FUNCTION_BLOCK TaskGUIFB (* JADE WORKER *)
  (* Standard: 61499-1 *)
  (* Version 1.0, 2014-04-22, Ahmed, Fraunhofer IGD *)
  (* Compiler header: package fb.gui; *)
  (* Compiler Java Sun JDK 1.5.0 *)
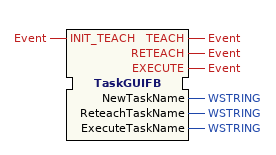
  EVENT_INPUT
    INIT_TEACH;
  END_EVENT
  EVENT_OUTPUT
    TEACH;
    RETEACH;
    EXECUTE;
  END_EVENT
  VAR_OUTPUT
    NewTaskName : WSTRING;
    ReteachTaskName : WSTRING;
    ExecuteTaskName : WSTRING;
  END_VAR
END_FUNCTION_BLOCK
